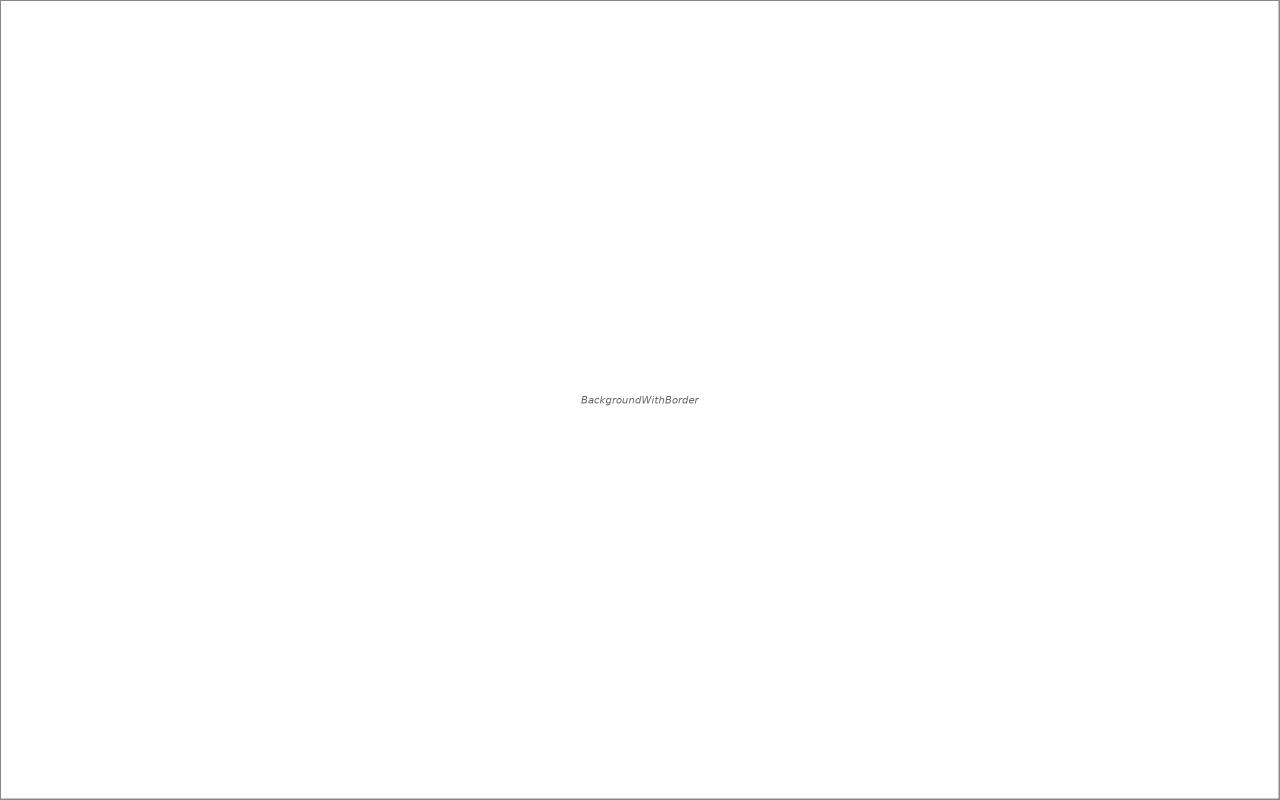
VISUALIZATION BaseScreen  // 1280x800
    Frame (0,0 1280x800)
        shows BackgroundWithBorder()
END_VISUALIZATION

(* stored: Version 1.1.0.1, ProductVersion 3.1.4024.9
   Visu BaseScreen: Id {4947af5d-5d50-4f16-ab4a-243dcb1607d8} *)
